// Mitsubishi GX Works2 project: DK_Thuan_Nghich_Tat_Sau5s   PLC: FX2N/FX2NC

PROGRAM MAIN
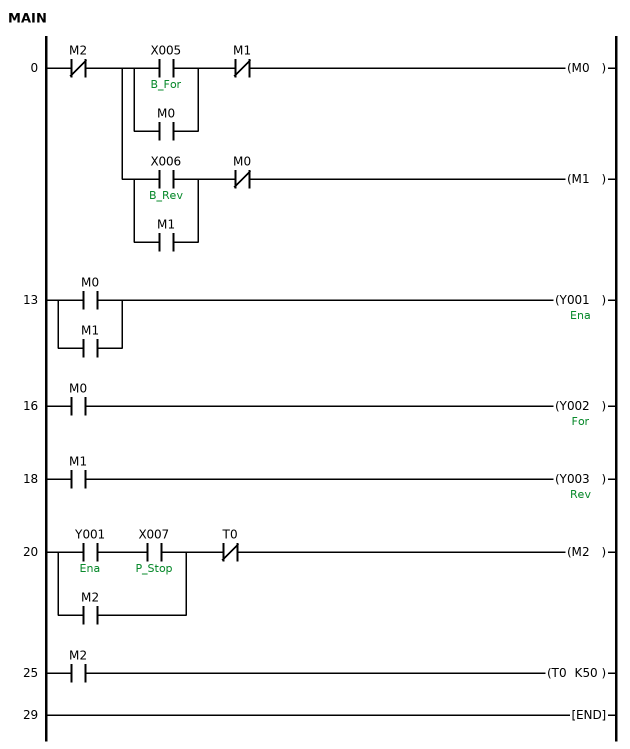
0     LDI     M2
      MPS
      LD      X005  ; B_For
      OR      M0
      ANB
      ANI     M1
      OUT     M0
      MPP
      LD      X006  ; B_Rev
      OR      M1
      ANB
      ANI     M0
      OUT     M1
13    LD      M0
      OR      M1
      OUT     Y001  ; Ena
16    LD      M0
      OUT     Y002  ; For
18    LD      M1
      OUT     Y003  ; Rev
20    LD      Y001  ; Ena
      AND     X007  ; P_Stop
      OR      M2
      ANI     T0
      OUT     M2
25    LD      M2
      OUT     T0 K50
29    END
END_PROGRAM
